FUNCTION_BLOCK DataPanel_MI_QX (* Output service interface function block for boolean output data *)
  (* Description: Copyright (c) 2014, 2015 fortiss GmbH This program and the accompanying materials are made available under the terms of the Eclipse Public License 2.0 which is available at https://www.eclipse.org/legal/epl-2.0/ SPDX-License-Identifier: EPL-2.0 *)
  (* Version 1.0, 2014-08-26, Waldemar Eisenmenger, fortiss GmbH *)
  (* Version 1.1, 2014-08-30, Alois Zoitl, fortiss GmbH *)
  (* Version 1.2, 2015-06-10, Monika Wenger, fortiss GmbH *)
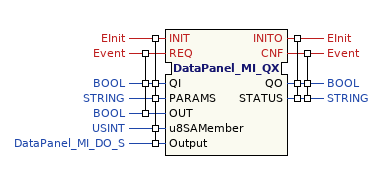
  EVENT_INPUT
    INIT : EInit WITH QI, PARAMS, u8SAMember, Output; (* Service Initialization *)
    REQ WITH QI, OUT; (* Service Request *)
  END_EVENT
  EVENT_OUTPUT
    INITO : EInit WITH QO, STATUS; (* Initialization Confirm *)
    CNF WITH QO, STATUS; (* Confirmation of Requested Service *)
  END_EVENT
  VAR_INPUT
    QI : BOOL; (* Event Input Qualifier *)
    PARAMS : STRING; (* Service Parameters *)
    OUT : BOOL; (* Output data to resource *)
    u8SAMember : USINT := MI::MI_00; (* Node SA 224..239 *)
    Output : DataPanel_MI_DO_S := DataPanel_MI_DO::Invalid; (* Identify the Output DigitalOutput_1A..8B and Input_Power_Port_5..8 *)
  END_VAR
  VAR_OUTPUT
    QO : BOOL; (* Event Output Qualifier *)
    STATUS : STRING; (* Service Status *)
  END_VAR
END_FUNCTION_BLOCK
